{attribute 'qualified_only'}
{attribute 'strict'}
{attribute 'to_string'}
TYPE E_ComponentTypes :
(
	// No entry
		NA			:= 0,
	// Actuators 
		Cylinder 	:= 10,
		Axis		:= 11,
		Heaters		:= 12,
	// Buttons 
		EstopButton	:= 20,
		EstopBumper	:= 21,	
		Pushbutton 	:= 22,
		Switch		:= 23,
	// I/O
		SafeIO		:= 30,
		Rio_Box		:= 31,
		Rio_Slot	:= 32,
		Encoder		:= 33,
		DiInput		:= 34,
		AnInput		:= 35,
		DiOutput	:= 36,
		AnOutput	:= 37,
	// Drive
		ServoDrive 	:= 40,
	// Operation
		HMI			:= 50,
		RemoteOS	:= 51,
		RemoteDB	:= 52,
	// Assemblies
		Assembly 	:= 60,
		SubAssembly	:= 61,
	// functions
		MainProgram		:= 100,
		StepProgram		:= 101,
		FunctionBlock	:= 102 
)UDINT;
END_TYPE

(* stored: Version 1.1.0.1, ProductVersion 3.1.4024.11
   EnumerationTextList E_ComponentTypes: Id {279e7338-601a-42f5-8e17-8ce44587bb9a} *)
